{attribute 'qualified_only'}
VAR_GLOBAL
	InterfaceManager_InstanceCounter :UINT;
END_VAR

(* stored: Version 1.1.0.1, ProductVersion 3.1.4024.6
   GVL _internal: Id {16aa3413-b429-0014-0c2f-56e4554e8f95} *)
